FUNCTION_BLOCK E_DELAY_V_D_B (* Basic Function Block Type *)
  (* Standard: 61499-2 *)
  (* Version 0.0, 6/13/2026, Schneider Electric, Template *)
  PACKAGE SE.Nereda;
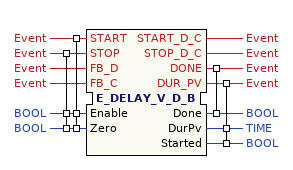
  EVENT_INPUT
    START WITH Enable, Zero;
    STOP WITH Enable, Zero;
    FB_D;
    FB_C;
  END_EVENT
  EVENT_OUTPUT
    START_D_C;
    STOP_D_C;
    DONE WITH Done;
    DUR_PV WITH DurPv, Started;
  END_EVENT
  VAR_INPUT
    Enable : BOOL;
    Zero : BOOL;
  END_VAR
  VAR_OUTPUT
    Done : BOOL;
    DurPv : TIME;
    Started : BOOL;
  END_VAR
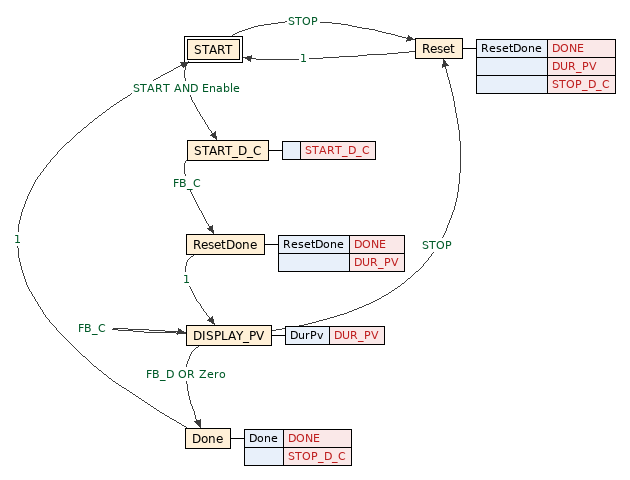
  EC_STATES
    START; (* Initial State *)
    START_D_C : -> START_D_C;
    DISPLAY_PV : DurPv -> DUR_PV;
    ResetDone : ResetDone -> DONE, -> DUR_PV;
    Done : Done -> DONE, -> STOP_D_C;
    Reset : ResetDone -> DONE, -> DUR_PV, -> STOP_D_C;
  END_STATES
  EC_TRANSITIONS
    START TO START_D_C := START AND Enable;
    START_D_C TO ResetDone := FB_C;
    ResetDone TO DISPLAY_PV := 1;
    DISPLAY_PV TO Reset := STOP;
    DISPLAY_PV TO Done := FB_D OR Zero;
    DISPLAY_PV TO DISPLAY_PV := FB_C;
    Done TO START := 1;
    START TO Reset := STOP;
    Reset TO START := 1;
  END_TRANSITIONS
  ALGORITHM ResetDone IN ST:
;
Done := FALSE;
DurPv := T#0s;
FB_C := FALSE;
Started := FALSE;
  END_ALGORITHM
  ALGORITHM DurPv IN ST:
;
DurPv := DurPv + T#1s;
Started := TRUE;
  END_ALGORITHM
  ALGORITHM Done IN ST:
;
Done := TRUE;
Started := FALSE;
  END_ALGORITHM
END_FUNCTION_BLOCK
